FUNCTION_BLOCK SIntComparer EXTENDS Object IMPLEMENTS IComparer
VAR
	_ClassName : STRING := __POUNAME();
END_VAR

{attribute 'monitoring' := 'call'}
PROPERTY ClassName : STRING
GET
ClassName := _ClassName;
END_GET
END_PROPERTY

{attribute "object_name" := "Compare"}
METHOD Compare : COMPARISION_RESULT
VAR_INPUT
	left : __SYSTEM.AnyType;
	right : __SYSTEM.AnyType;
END_VAR
VAR
	leftPointer : POINTER TO SINT; 
	rightPointer : POINTER TO SINT; 
END_VAR
IF left.pValue = 0 AND right.pValue = 0 THEN
	Compare := COMPARISION_RESULT.FIRST_EQUAL_TO_SECOND;
	RETURN;
END_IF

IF left.pValue = 0 THEN
	Compare := COMPARISION_RESULT.FIRST_LESS_THAN_SECOND;
	RETURN;	
END_IF

IF right.pValue = 0 THEN
	Compare := COMPARISION_RESULT.FIRST_GREATER_THAN_SECOND;
	RETURN;	
END_IF

leftPointer := left.pValue;
rightPointer := right.pValue;

IF leftPointer^ < rightPointer^ THEN
	Compare := COMPARISION_RESULT.FIRST_LESS_THAN_SECOND;
ELSIF leftPointer^ > rightPointer^ THEN
	Compare := COMPARISION_RESULT.FIRST_GREATER_THAN_SECOND;
ELSE
	Compare := COMPARISION_RESULT.FIRST_EQUAL_TO_SECOND;	
END_IF
END_METHOD

{attribute 'monitoring' := 'call'}
PROPERTY Size : ULINT
GET
Size := XSIZEOF(THIS^);
END_GET
END_PROPERTY

END_FUNCTION_BLOCK

(* stored: Version 1.1.0.1
   POU SIntComparer: Id {af8c7cfb-00c0-4dc2-8e54-aab52ae9c88f}, SpecialFunc None
   Property ClassName: Id {75615a5f-d5f9-4764-bc4d-e8e41ccf2940}
   Get Get: Id {38759394-2fc9-442d-a89a-9ec371c3b58d}
   Method Compare: Id {3092262e-9e30-4822-bd4f-4a148b4b0ad3}
   Property Size: Id {4eaf3d61-4042-40b3-90d2-9bcf14e6138c}
   Get Get: Id {8af84884-ba37-4735-9f1d-76e63b4c0147} *)
